(* CoDeSys 2.3.9.37 project: Cap3_1.pro *)
(* Libraries: Standard.lib 4.10.05 12:14:46 *)

(* POU PLC_PRG, LD *)
PROGRAM PLC_PRG
VAR
   A  : BOOL;
   B : BOOL;
   C : BOOL;
   Sal : BOOL;
END_VAR
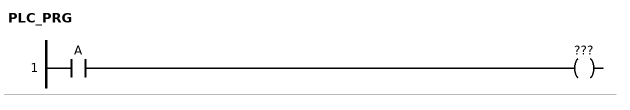
_LD_ (* Ladder Diagram *)
NETWORK 1
	[A] --- (???)
_END_LD_
END_PROGRAM

(* Visualisation Ejer1
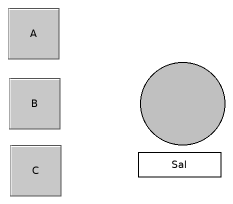
button at (66,37)-(117,88): text "A"; toggles PLC_PRG.A
button at (67,107)-(118,158): text "B"; toggles PLC_PRG.B
button at (68,174)-(119,225): text "C"; toggles PLC_PRG.C
ellipse at (198,91)-(283,174): alarm colour if PLC_PRG.Sal
rectangle at (196,181)-(279,206): text "Sal"
*)
